(* POU Plant_Objects/obj_TPV_SENS, ST *)
FUNCTION_BLOCK obj_TPV_SENS
(* === TEMPERATURE PROBE FROM ANALOG INPUT ===
   v1.0[16/04/05] - Versioning
*)
VAR_INPUT
	(* Settings *)
	ID				: BYTE;
	PuntoMinX		: INT;			(* Parametri per la scalatura *)
	PuntoMaxX		: INT;
	PuntoMinY		: REAL;
	PuntoMaxY		: REAL;
	Decimali		: BYTE:=1;
	SogliaHH		: WORD;			(* Soglia per segnalazione Allarme Extra Range in alto - Solitamente sondo in CC *)
	SogliaHL		: WORD;			(* Soglia per segnalazione Allarme Extra Range in Basso - Solitamente sondo Aperta *)
	SogliaWH		: REAL;			(* Soglia per segnalazione Warning  in alto  *)
	SogliaWL		: REAL;    		(* Soglia per segnalazione Warning in basso  *)
	TAP				: INT:=2000;	(* Filtro in msec *)
	INITEV			: BOOL:= TRUE;	(* Generate init OK event *)
	(* Physical input *)
	AI_INPUT		: WORD;    		(* Sensor analog input *)
END_VAR
VAR_OUTPUT
	WRN				: BOOL;	(* Segnalazione Warning *)
	ERR				: BOOL; (* Segnalazione Errore *)
	ValoreScalato	: INT;
	(* Status *)
	Status_Log	: BYTE;
	Status_Vis 	: DWORD;
END_VAR
VAR
	SegnaleHH	: BOOL;
	SegnaleHL	: BOOL;
	SegnaleOK	: BOOL;
	SegnaleWH	: BOOL;
	SegnaleWL	: BOOL;
    FiltroWRN	: TON;
    FiltroOK	: TON;
    FiltroERR	: TON;
END_VAR
(* Verifico che le variabile letta dall'ingresso Analogico  sia dentro i range
ATTENZIONE I LIMITI SPESSO SONO IN WORD VERIFICA  TABELLA MANUALE WAGO  *)

SegnaleHH:=(AI_INPUT>=SogliaHH);
SegnaleHL:=(AI_INPUT<=SogliaHL);
SegnaleOK:=NOT (SegnaleHH OR SegnaleHL);

(* Linerarizzo il segnale di ingresso e la converto in unita ingegneristiche *)
ValoreScalato:=LINEAR_BAD(PuntoMinX, PuntoMaxX, AI_INPUT, PuntoMinY, PuntoMaxY, Decimali);


IF SegnaleOK  THEN
	(*  Verifica  e segnalazione Warning *)
	SegnaleWH:=(ValoreScalato>SogliaWH*(EXPT(10, Decimali)));
	SegnaleWL:=(ValoreScalato<SogliaWL*(EXPT(10, Decimali)));

	FiltroWRN( IN:=(SegnaleWH OR SegnaleWL), PT:=INT_TO_TIME(TAP) );    (* Filtro su LOG *)
	IF  FiltroWRN.Q THEN     (* Condizione di WARNING *)
		IF NOT WRN THEN
			WRN:=TRUE;
			LogEv(EL_Wrn,EO_TPV,ID,SEL(ValoreScalato<=SogliaWL,3,2),INT_TO_STRING(ValoreScalato));
		END_IF
	END_IF

    IF (INITEV OR WRN OR ERR) AND NOT FiltroWRN.Q THEN
		FiltroWRN(IN:=FALSE  , PT:=INT_TO_TIME(TAP));    (* Resetto il Filtro su LOG WRN  *)
		FiltroERR(IN:=FALSE  , PT:=INT_TO_TIME(TAP));    (* Resetto il Filtro su LOG ERR *)
		INITEV:=FALSE; ERR:=FALSE; WRN:=FALSE;
		LogEv(EL_Log,EO_TPV,ID,1,'');
	END_IF

	Status_Vis:=16#20F020;    (* Indicazione WEB Visu Sonda OK *)
ELSE
	FiltroERR(IN:=TRUE  , PT:= INT_TO_TIME(TAP) );    (* Filtro su LOG *)
	IF  FiltroERR.Q THEN     (* Condizione di WARNING *)
		IF NOT ERR THEN
			ERR:=TRUE;
			IF SegnaleHH THEN LogEv(EL_Alarm,EO_TPV,ID,6,INT_TO_STRING(ValoreScalato));END_IF;
			IF SegnaleHL THEN LogEv(EL_Alarm,EO_TPV,ID,4,INT_TO_STRING(ValoreScalato));END_IF;
		END_IF
	END_IF

	Status_Vis:=16#2020F0;   (* Indicazione WEB Visu Sonda KO *)
END_IF
END_FUNCTION_BLOCK

(* POU Plant_Objects/obj_TPV_SENS2, ST *)
FUNCTION_BLOCK obj_TPV_SENS2
(* === TEMPERATURE PROBE FROM ANALOG INPUT ===
   v2.0[17/04/05] - Versioning
*)
VAR_INPUT
	(* Settings *)
	ID				: BYTE;
	TAP				: BYTE:=4;	   (* Consecutive checks filter *)
	INITEV			: BOOL:= TRUE; (* Generate init OK event *)
	IN_EMIN			: INT :=-2000; (* Low error limit *)
	IN_WMIN			: INT := -550; (* Low warning value *)
	IN_WMAX			: INT :=  900; (* High warning value *)
	IN_EMAX			: INT := 8500; (* High error limit *)
	ERR_MIN_SHORT	: BOOL:= TRUE; (* TRUE  ==> EMIN=Short        , EMAX=Disconnected
									  FALSE ==> EMIN=Disconnected , EMAX=Short 		 *)
	SCALE_LO_IN		: WORD;
	SCALE_LO_OUT	: INT;
	SCALE_HI_IN		: WORD;
	SCALE_HI_OUT	: INT;

	(* Physical input *)
	IN				: WORD;			(* Sensor analog input *)

	(* Settings *)
	PuntoMinX		: INT;			(* Parametri per la scalatura *)
	PuntoMaxX		: INT;
	PuntoMinY		: REAL;
	PuntoMaxY		: REAL;

	SogliaHH		: WORD;			(* Soglia per segnalazione Allarme Extra Range in alto - Solitamente sondo in CC *)
	SogliaHL		: WORD;			(* Soglia per segnalazione Allarme Extra Range in Basso - Solitamente sondo Aperta *)
	SogliaWH		: REAL;			(* Soglia per segnalazione Warning  in alto  *)
	SogliaWL		: REAL;    		(* Soglia per segnalazione Warning in basso  *)
END_VAR
VAR_OUTPUT
	OUT			: INT;
	OUT_VALID	: BOOL;
	(* Status *)
	Status_Log	: BYTE;
	Status_Vis 	: DWORD;
END_VAR
VAR
	SegnaleHH	: BOOL;
	SegnaleHL	: BOOL;
	SegnaleOK	: BOOL;
	SegnaleWH	: BOOL;
	SegnaleWL	: BOOL;
    FiltroWRN	: TON;
    FiltroOK	: TON;
    FiltroERR	: TON;
END_VAR
(* Verifico che le variabile letta dall'ingresso Analogico  sia dentro i range
ATTENZIONE I LIMITI SPESSO SONO IN WORD VERIFICA  TABELLA MANUALE WAGO  *)

SegnaleHH:=(AI_INPUT>=SogliaHH);
SegnaleHL:=(AI_INPUT<=SogliaHL);
SegnaleOK:=NOT (SegnaleHH OR SegnaleHL);

(* Linerarizzo il segnale di ingresso e la converto in unita ingegneristiche *)
OUT:=LINEAR_BAD(PuntoMinX, PuntoMaxX, AI_INPUT, PuntoMinY, PuntoMaxY, Decimali);


IF SegnaleOK  THEN
	(*  Verifica  e segnalazione Warning *)
	SegnaleWH:=(OUT > SogliaWH*(EXPT(10, Decimali)));
	SegnaleWL:=(OUT < SogliaWL*(EXPT(10, Decimali)));

	FiltroWRN( IN:=(SegnaleWH OR SegnaleWL), PT:=INT_TO_TIME(TAP) );    (* Filtro su LOG *)
	IF  FiltroWRN.Q THEN     (* Condizione di WARNING *)
		IF NOT WRN THEN
			WRN:=TRUE;
			LogEv(EL_Wrn,EO_TPV,ID,SEL(ValoreScalato<=SogliaWL,3,2),INT_TO_STRING(ValoreScalato));
		END_IF
	END_IF

    IF (INITEV OR WRN OR ERR) AND NOT FiltroWRN.Q THEN
		FiltroWRN(IN:=FALSE  , PT:=INT_TO_TIME(TAP));    (* Resetto il Filtro su LOG WRN  *)
		FiltroERR(IN:=FALSE  , PT:=INT_TO_TIME(TAP));    (* Resetto il Filtro su LOG ERR *)
		INITEV:=FALSE; ERR:=FALSE; WRN:=FALSE;
		LogEv(EL_Log,EO_TPV,ID,1,'');
	END_IF

	Status_Vis:=16#20F020;    (* Indicazione WEB Visu Sonda OK *)
ELSE
	FiltroERR(IN:=TRUE  , PT:= INT_TO_TIME(TAP) );    (* Filtro su LOG *)
	IF  FiltroERR.Q THEN     (* Condizione di WARNING *)
		IF NOT ERR THEN
			ERR:=TRUE;
			IF SegnaleHH THEN LogEv(EL_Alarm,EO_TPV,ID,6,INT_TO_STRING(ValoreScalato));END_IF;
			IF SegnaleHL THEN LogEv(EL_Alarm,EO_TPV,ID,4,INT_TO_STRING(ValoreScalato));END_IF;
		END_IF
	END_IF

	Status_Vis:=16#2020F0;   (* Indicazione WEB Visu Sonda KO *)
END_IF
END_FUNCTION_BLOCK

(* POU PLC_WDT, ST *)
FUNCTION PLC_WDT: DWORD VAR_INPUT dwEvent: DWORD; dwFilter: DWORD; dwOwner: DWORD; END_VAR
LogEv(EL_AlarmStop,EO_SYS,1,10,'Watchdog');
END_FUNCTION

(* POU Utils Functions/RAW16TOHEXSTR, ST *)
FUNCTION RAW16TOHEXSTR : STRING(128)
VAR_INPUT
	pData: POINTER TO BYTE;
	DataLen: BYTE;
END_VAR
VAR
	pt: POINTER TO BYTE;
	xl: BYTE;
END_VAR
pt:=ADR(RAW16TOHEXSTR);
xl:=0;

WHILE DataLen>0 AND xl<120 DO

	pData:=pData+1;

	pt^ := (pData^ / 16#10) + 48 + (((pData^ / 16#10)/10)*7);
	pt:=pt+1;
	pt^ := (pData^ AND 16#0F)  + 48 + (((pData^ AND 16#0F)/10)*7);
	pt:=pt+1;

	pData:=pData-1;

	pt^ := (pData^ / 16#10) + 48 + (((pData^ / 16#10)/10)*7);
	pt:=pt+1;
	pt^ := (pData^ AND 16#0F)  + 48 + (((pData^ AND 16#0F)/10)*7);
	pt:=pt+1;

	xl:=xl+4;

	DataLen:=DataLen-2;
	pData:=pData+2;

END_WHILE

pt^:=0;
END_FUNCTION

(* POU Utils Functions/RAWTOHEX, ST *)
FUNCTION RAWTOHEX : WORD
VAR_INPUT
	pData: POINTER TO BYTE;
	DataLen: WORD;
	pString: POINTER TO BYTE;
END_VAR
VAR
	xl: WORD;
END_VAR
xl:=0;

WHILE DataLen>0 DO

	pString^ := (pData^ / 16#10) + 48 + (((pData^ / 16#10)/10)*7);
	pString:=pString+1;
	pString^ := (pData^ AND 16#0F)  + 48 + (((pData^ AND 16#0F)/10)*7);
	pString:=pString+1;
	pData:=pData+1;
	DataLen:=DataLen-1;
	xl:=xl+2;

END_WHILE

(*pString^:=0;*)

RAWTOHEX:=xl;
END_FUNCTION

(* POU Utils Functions/RAWTOHEXSTR, ST *)
FUNCTION RAWTOHEXSTR : STRING(128)
VAR_INPUT
	pData: POINTER TO BYTE;
	DataLen: BYTE;
END_VAR
VAR
	pt: POINTER TO BYTE;
	xl: BYTE;
END_VAR
pt:=ADR(RAWTOHEXSTR);

xl:=2;

WHILE DataLen>0 AND xl<128 DO

	pt^ := (pData^ / 16#10) + 48 + (((pData^ / 16#10)/10)*7);
	pt:=pt+1;
	pt^ := (pData^ AND 16#0F)  + 48 + (((pData^ AND 16#0F)/10)*7);
	pt:=pt+1;

	xl:=xl+2;

	DataLen:=DataLen-1;
	pData:=pData+1;

END_WHILE

pt^:=0;
END_FUNCTION

(* POU Utils/RTC_Update, ST *)
FUNCTION RTC_Update : BOOL
VAR
	T: DT;
	TS: STRING;
	TS2: STRING;
	Hour: BYTE;
	Minute: BYTE;
END_VAR
(* Get RTC time *)
T:=SysRtcGetTime(TRUE);
Sys.Time_CT_DT:=T;
(* Calculate variables *)
TS:=DT_TO_STRING(T);
Sys.Time_LogString:=DELETE(STR:=TS, LEN:=3, POS:=1);
TS2:=MID(STR:=TS, LEN:=4, POS:= 4); Sys.Time_Year 	:=STRING_TO_WORD(TS2);
TS2:=MID(STR:=TS, LEN:=2, POS:= 9); Sys.Time_Month	:=STRING_TO_BYTE(TS2);
TS2:=MID(STR:=TS, LEN:=2, POS:=12); Sys.Time_Day  	:=STRING_TO_BYTE(TS2);
Sys.Time_CT_Day:=(32*(Sys.Time_Month-1)+Sys.Time_Day-1);
TS2:=MID(STR:=TS, LEN:=2, POS:=15); Hour			:=STRING_TO_BYTE(TS2);
TS2:=MID(STR:=TS, LEN:=2, POS:=18); Minute		 	:=STRING_TO_BYTE(TS2);
Sys.Time_CT_Quarter:=Hour*4+(Minute/15);
END_FUNCTION

(* POU Utils Functions/TONOF, ST *)
FUNCTION_BLOCK TONOF
VAR_INPUT
	IN		: BOOL;
	PT_ON	: TIME; (* time to pass, before OUT is set *)
	PT_OF	: TIME; (* time to pass, before OUT is reset *)
END_VAR
VAR_OUTPUT
	OUT		: BOOL;
END_VAR
VAR
	timer	: TON;
END_VAR
IF IN<>OUT THEN
	timer(IN:=TRUE,PT:=SEL(IN,PT_OF,PT_ON));
	IF timer.Q THEN OUT:=IN; END_IF
ELSE
	timer(IN:=FALSE);
END_IF
END_FUNCTION_BLOCK

(* Visualisation PLC_VISU
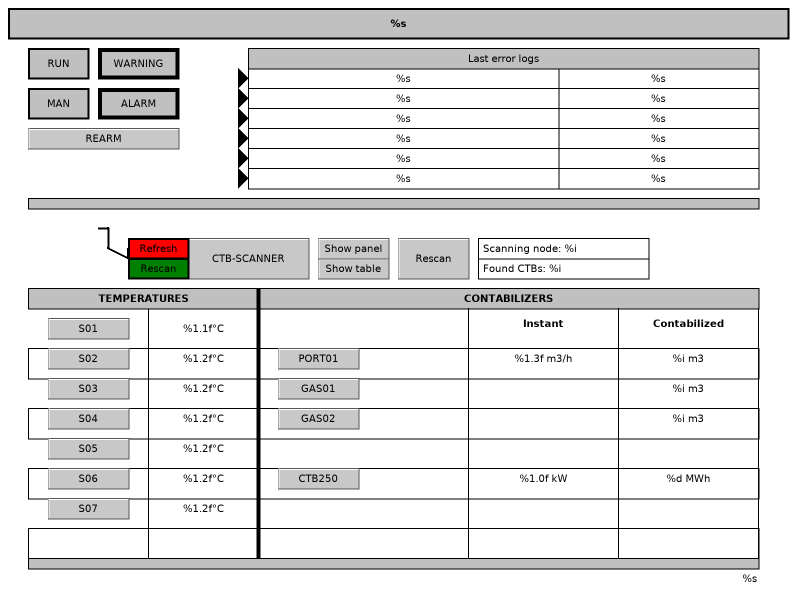
button at (50,350)-(131,371): text "S02"
rectangle at (520,570)-(761,591): text "%s"; shows Sys.Time_LogString
rectangle at (10,10)-(791,41): text "%s"; shows .Plant_NAME
rectangle at (160,350)-(251,371): text "%1.2f°C"; shows INT_TO_REAL(.TPV02.ValoreScalato)/(.TPV02.Decimali*10)
rounded rectangle at (30,50)-(91,81): text "RUN"; alarm colour if NOT Mode_Manual; runs INTERN ASSIGN Mode_Manual:=(FALSE)
rounded rectangle at (30,90)-(91,121): text "MAN"; alarm colour if Mode_Manual; runs INTERN ASSIGN Mode_Manual:=(TRUE)
button at (190,240)-(311,281): text "CTB-SCANNER"
rectangle at (100,90)-(181,121): text "ALARM"; alarm colour if Sys.Alarm; runs INTERN ASSIGN Mode_Manual:=(FALSE)
rectangle at (100,50)-(181,81): text "WARNING"; alarm colour if Sys.Warning; runs INTERN ASSIGN Mode_Manual:=(TRUE)
button at (30,130)-(181,151): text "REARM"; runs INTERN ASSIGN Sys.Alarm:=(FALSE);INTERN ASSIGN Sys.Warning:=(FALSE)
button at (50,320)-(131,341): text "S01"
rectangle at (160,320)-(251,341): text "%1.1f°C"; shows INT_TO_REAL(.TPV01.IN)/10
button at (50,380)-(131,401): text "S03"
rectangle at (160,380)-(251,401): text "%1.2f°C"; shows INT_TO_REAL(.TPV03.ValoreScalato)/(.TPV03.Decimali*10)
button at (50,410)-(131,431): text "S04"
rectangle at (160,410)-(251,431): text "%1.2f°C"; shows INT_TO_REAL(.TPV04.ValoreScalato)/(.TPV04.Decimali*10)
button at (50,440)-(131,461): text "S05"
rectangle at (160,440)-(251,461): text "%1.2f°C"; shows INT_TO_REAL(.TPV05.ValoreScalato)/(.TPV05.Decimali*10)
button at (50,470)-(131,491): text "S06"
rectangle at (160,470)-(251,491): text "%1.2f°C"; shows INT_TO_REAL(.TPV06.ValoreScalato)/(.TPV06.Decimali*10)
button at (50,500)-(131,521): text "S07"
rectangle at (160,500)-(251,521): text "%1.2f°C"; shows INT_TO_REAL(.TPV07.ValoreScalato)/(.TPV07.Decimali*10)
rectangle at (30,290)-(261,311): text "TEMPERATURES"
rectangle at (260,290)-(761,311): text "CONTABILIZERS"
button at (280,350)-(361,371): text "PORT01"
rectangle at (480,350)-(611,371): text "%1.3f m3/h"; shows DINT_TO_REAL(.PORT01.ValoreScalato)/1000
rectangle at (470,310)-(621,341): text "Instant"
rectangle at (630,350)-(751,371): text "%i m3"; shows .PortataTotalePORT01
rectangle at (620,310)-(761,341): text "Contabilized"
button at (280,380)-(361,401): text "GAS01"
button at (280,410)-(361,431): text "GAS02"
rectangle at (630,380)-(751,401): text "%i m3"; shows .PortataTotaleGAS01
rectangle at (630,410)-(751,431): text "%i m3"; shows .PortataTotaleGAS02
rectangle at (560,70)-(761,91): text "%s"; shows Sys.LastLogs_Msg[0]
polygon at (240,170)-(250,190): invisible if Sys.LastLogs_Idx<>0
rectangle at (560,90)-(761,111): text "%s"; shows Sys.LastLogs_Msg[1]
polygon at (240,70)-(250,90): invisible if Sys.LastLogs_Idx<>1
rectangle at (560,110)-(761,131): text "%s"; shows Sys.LastLogs_Msg[2]
polygon at (240,90)-(250,110): invisible if Sys.LastLogs_Idx<>2
rectangle at (560,130)-(761,151): text "%s"; shows Sys.LastLogs_Msg[3]
polygon at (240,110)-(250,130): invisible if Sys.LastLogs_Idx<>3
rectangle at (560,150)-(761,171): text "%s"; shows Sys.LastLogs_Msg[4]
polygon at (240,130)-(250,150): invisible if Sys.LastLogs_Idx<>4
rectangle at (560,170)-(761,191): text "%s"; shows Sys.LastLogs_Msg[5]
polygon at (240,150)-(250,170): invisible if Sys.LastLogs_Idx<>5
rectangle at (250,70)-(561,91): text "%s"; shows Sys.LastLogs_Dat[0]
rectangle at (250,90)-(561,111): text "%s"; shows Sys.LastLogs_Dat[1]
rectangle at (250,110)-(561,131): text "%s"; shows Sys.LastLogs_Dat[2]
rectangle at (250,130)-(561,151): text "%s"; shows Sys.LastLogs_Dat[3]
rectangle at (250,150)-(561,171): text "%s"; shows Sys.LastLogs_Dat[4]
rectangle at (250,170)-(561,191): text "%s"; shows Sys.LastLogs_Dat[5]
rectangle at (250,50)-(761,71): text "Last error logs"
button at (400,240)-(471,281): text "Rescan"; runs INTERN ASSIGN CTBSCAN01.Rescan:=(TRUE)
rectangle at (130,240)-(191,261): text "Refresh"; alarm colour if .CTBSCAN01.Refresh; toggles .CTBSCAN01.Refresh
rectangle at (130,260)-(191,281): text "Rescan"; alarm colour if .CTBSCAN01.Rescan
rectangle at (480,260)-(651,281): text "Found CTBs: %i"; shows .CTBSCAN01.ConnectedCTBs
rectangle at (480,240)-(651,261): text "Scanning node: %i"; shows .CTBSCAN01.cnt
rectangle at (480,470)-(611,491): text "%1.0f kW"; shows .CTB250.POWER_KW
rectangle at (630,470)-(751,491): text "%d MWh"; shows .CTB250.ENERGY/100
button at (280,470)-(361,491): text "CTB250"
button at (320,260)-(391,281): text "Show table"; opens VIS_CTBSCAN01
button at (320,240)-(391,261): text "Show panel"; opens VIS_CTBSCAN01_PANEL
12 more shapes without text or variables
13 elements of other kinds (tables, trends, ...) not read
*)

(* Visualisation VIS_CTBSCAN01
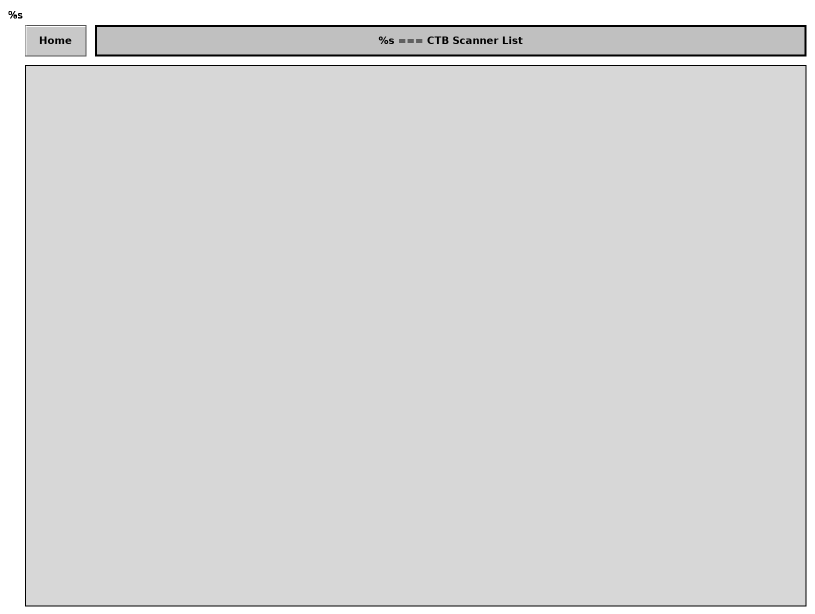
rectangle at (0,0)-(0,0): text "%s"; shows CTBSCAN01.VisuDatiMbus[INDEX].sdNodoPresente; alarm colour if CTBSCAN01.NodoMBusPresente[INDEX]; editable
rectangle at (0,0)-(0,0): text "%s"; shows CTBSCAN01.VisuDatiMbus[INDEX].sdEnergia
rectangle at (0,0)-(0,0): text "%s"; shows CTBSCAN01.VisuDatiMbus[INDEX].sdPotenza
rectangle at (0,0)-(0,0): text "%s"; shows CTBSCAN01.VisuDatiMbus[INDEX].sdVolume
rectangle at (0,0)-(0,0): text "%s"; shows CTBSCAN01.VisuDatiMbus[INDEX].sdFlow
rectangle at (0,0)-(0,0): text "%s"; shows CTBSCAN01.VisuDatiMbus[INDEX].sdTempIngresso
rectangle at (0,0)-(0,0): text "%s"; shows CTBSCAN01.VisuDatiMbus[INDEX].sdTempaUscita
rectangle at (0,0)-(0,0): text "%s"; shows CTBSCAN01.VisuDatiMbus[INDEX].sdTempDelta
rectangle at (80,10)-(791,41): text "%s === CTB Scanner List"; shows .Plant_NAME
button at (10,10)-(71,41): text "Home"; opens PLC_VISU
1 more shapes without text or variables
*)

(* Visualisation VIS_CTBSCAN01_PANEL
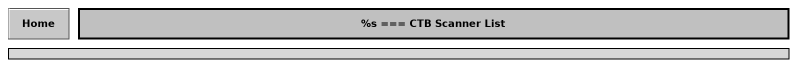
rectangle at (80,10)-(791,41): text "%s === CTB Scanner List"; shows .Plant_NAME
button at (10,10)-(71,41): text "Home"; opens PLC_VISU
1 more shapes without text or variables
250 elements of other kinds (tables, trends, ...) not read
*)
